Universal Robots PolyScope program: MQTT_Main.urp

Program MQTT_Main (installation=default directory=/ursim/programs/MQTT createdIn=5.13.0 lastSavedIn=5.16.0 robotSerialNumber=20195599999)
Calibrated DH parameters: a=[0, -0.425, -0.3922, 0, 0, 0]; d=[0.1625, 0, 0, 0.1333, 0.0997, 0.0996]; alpha=[1.570796, 0, 0, 1.570796, -1.570796, 0]; deltaTheta=[0, 0, 0, 0, 0, 0]
InitVariablesNode variables(variable(name=cmd_name, expression=""), variable(name=object, expression=" "), variable(name=params, expression=" "), variable(name=topic_order, expression="robot/order"))
BeforeStart
  Script file /ursim/programs/MQTT/json.script
    | ###
    | # summary: This function is used to split a string into an array of substrings with a delimiter
    | # @param str :string the string to split
    | # @param delimiter :string the caracter to split the string
    | # @param debug :bool activ message debug
    | ###
    | MAX_VARIABLES = 100
    | def str_split(str, delimiter, debug=False):
    |   result = make_list(0, "", MAX_VARIABLES) # Arrays to stock the result max 10 variables
    |   start = 0  # Position to start the search
    |   end_deli = str_find(str, delimiter) #Find the first delimiter
    | 
    |   # While a delimiter is found
    |   while end_deli != -1:
    |     if result.excess_capacity() == 0:
    |       if debug:
    |         textmsg("Number of variables exceeded")
    |       end
    |       return result
    |     end
    | 
    |     # Extraction of the substring between the start and the delimiter
    |     substring = str_sub(str, start, end_deli - start)
    |     result.append(substring)
    | 
    |     # Update the start position and the end delimiter
    |     str = str_sub(str, end_deli + str_len(delimiter), str_len(str))
    |     end_deli = str_find(str, delimiter)
    |   end
    | 
    |   # Add the last substring
    |   if result.excess_capacity() > 0:
    |     result.append(str)
    |   elif debug:
    |     textmsg("Number of variables exceeded")
    |   end
    | 
    |   if debug:
    |     textmsg("Result: " + result.to_string())
    |   end
    |   return result
    | end
    | 
    | 
    | ###
    | # summary: This function to return the value of a variable in a JSON string function only with string type
    | # @param json_string :string the json payload
    | # @param variable :string the variable the function needs to find
    | # @param debug :bool activ message debug
    | ###
    | def value_json_string(json_string, variable, type="str",debug=False):
    |   #Verify the json string is not empty (2 brackets at minimal)
    |   if str_len(json_string) < 2:
    |     if debug:
    |       textmsg("The JSON string is empty or invalid")
    |     end
    |     if(type == "int"):
    |       return 0
    |     end
    |     return " "
    |   end
    | 
    |   json_string = str_sub(json_string, 1, str_len(json_string) - 2) #Cut the first and last bracket
    |   variable_array = str_split(json_string, ",", debug) #Split the json string into an array of variables
    | 
    |   idx = 0 #Index of the array
    |   len_var_array = variable_array.length() #Length of the array
    | 
    |   #While the index is less than the length of the array
    |   while idx < len_var_array:
    | 
    |     find = str_find(variable_array[idx], variable) #Find the variable in the array
    |     if find > 0: #If the variable is found
    |       if debug:
    |         textmsg("Variable found")
    |       end
    |       value = str_split(variable_array[idx], ":")[1] #Split the variable to get the value
    |       if str_find(value, "'")>0: #If the value is a string
    |         return str_sub(value, 2, str_len(value) - 3) #Return the value without the quotes
    |       end
    |       if(type == "int"):
    |         return to_num(value)
    |       end
    |       return value
    |     end
    |     idx = idx + 1
    |   end
    |   if(type == "int"):
    |     return 0
    |   end
    |   return " "
    | end
  mqtt_init_state := mqtt_initialize_anonymous("mosquitto", 1883)
  mqtt_con_state := mqtt_connect()
  mqtt_sub_state := mqtt_subscribe(topic_order)
  old_payload := "NG-CODE-071"
  payload := "NG-CODE-071"
  MoveJ speed 60 deg/s, acceleration 80 deg/s^2 (useActiveTCP=true) feature=Base
    Waypoint waiting_point: TCP in base x=492.803 y=288.649 z=418.324 mm, rx=2.6568 ry=-1.6608 rz=-0.0199 rad; joints [192.415, -98.238, 124.325, -115.253, -89.954, -13.481] deg
Robot Program (runOnlyOnce=false)
  Wait Condition expression=payload != old_payload
  Wait Sleep waitTime=0.1
  If cmd_name == "Move"
    params := mqtt_get_json_message(topic_order, "params", params)
    Call Move_program
  ElseIf cmd_name == "Pickup"
    params := mqtt_get_json_message(topic_order, "params", params)
    Call Pickup_program
  ElseIf cmd_name == "Place"
    Call Place_program
  ElseIf cmd_name == "Rotate"
    Call Rotate_program
  old_payload := payload
SubProgram -> Rotate_program
Thread Thread_1 (runOnlyOnce=false)
  Loop Forever
    Wait Sleep waitTime=0.1
    payload := mqtt_get_message("robot/order")
    If payload != old_payload
      cmd_name := mqtt_get_json_message(topic_order, "name", cmd_name)
      If cmd_name=="Stop" (checkContinuously=true)
        Popup Warning (haltProgram=false message=Program Stop inputType=Text)
        Halt
SubProgram  [hidden by the author, left out]
SubProgram  [hidden by the author, left out]
SubProgram  [hidden by the author, left out]
SubProgram Move_program [hidden by the author, left out]
SubProgram Pickup_program [hidden by the author, left out]
SubProgram Place_program [hidden by the author, left out]
SubProgram Rotate_program (keepSynchronizedWithDisk=false) programFile=/ursim/programs/MQTT/Rotate_program.urp
  Script file /ursim/programs/angle.script
    | pose_actuelle = get_actual_tcp_pose()
    | angle_rotation = d2r(angle)
    | rotation_z = p[0, 0, 0, 0, 0, angle_rotation]
    | nouvelle_pose = pose_trans(pose_actuelle, rotation_z)
    | movel(nouvelle_pose)
